SUBAPPLICATION F_AI_RAW_TO_PERCENT (* Analog-Rohwert (DWORD 0-4095, 12-bit ESP32-P4-ADC-Vollausschlag) linear in Prozent (REAL 0.0-100.0) umrechnen - keine physikalische Kalibrierung (folgt spaeter) *)
  (* Standard: 61499-2 *)
  (* Version 1.0, 2026-08-30, franz *)
  PACKAGE MyLib::sys;
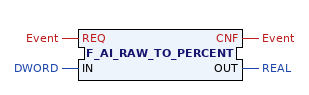
  EVENT_INPUT
    REQ; (* Normal Execution Request *)
  END_EVENT
  EVENT_OUTPUT
    CNF; (* Execution Confirmation *)
  END_EVENT
  VAR_INPUT
    IN : DWORD; (* Analog-Rohwert 0-4095 (12 bit, logiBUS_AI_ID/_IDA.IN) *)
  END_VAR
  VAR_OUTPUT
    OUT : REAL; (* Prozent 0.0-100.0, linear raw/4095*100, keine physikalische Einheit *)
  END_VAR
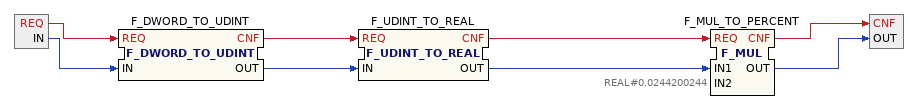
  FBS
    F_DWORD_TO_UDINT : iec61131::conversion::F_DWORD_TO_UDINT;
    F_UDINT_TO_REAL : iec61131::conversion::F_UDINT_TO_REAL;
    F_MUL_TO_PERCENT : iec61131::arithmetic::F_MUL(IN2 := REAL#0.0244200244);
  END_FBS
  EVENT_CONNECTIONS
    REQ TO F_DWORD_TO_UDINT.REQ;
    F_DWORD_TO_UDINT.CNF TO F_UDINT_TO_REAL.REQ;
    F_UDINT_TO_REAL.CNF TO F_MUL_TO_PERCENT.REQ;
    F_MUL_TO_PERCENT.CNF TO CNF;
  END_CONNECTIONS
  DATA_CONNECTIONS
    IN TO F_DWORD_TO_UDINT.IN;
    F_DWORD_TO_UDINT.OUT TO F_UDINT_TO_REAL.IN;
    F_UDINT_TO_REAL.OUT TO F_MUL_TO_PERCENT.IN1;
    F_MUL_TO_PERCENT.OUT TO OUT;
  END_CONNECTIONS
END_SUBAPPLICATION
